// TIA Portal V20 export
// export: Created 2026-04-11T06:02:30.0272566Z, ExportSetting WithDefaults, DisplayName Totally Integrated Automation Portal, DisplayVersion V20, DisplayName TIA Portal Openness, DisplayVersion V20, DisplayName TIA Portal Version Control Interface, DisplayVersion V20, DisplayName STEP 7 Professional, DisplayVersion V20, DisplayName STEP 7 Safety, DisplayVersion V20, DisplayName WinCC Basic/Comfort/Advanced, DisplayVersion V20, DisplayName WinCC Unified, DisplayVersion V20
TYPE "udtError_MicroMotion"
// stored: IsFailsafeCompliant false
   STRUCT
      ResetFailed { ExternalWritable := 'False'} : Bool;   // Can't reset MicroMotion
      FlowWithoutRequest { ExternalWritable := 'False'} : Bool;   // Flow detected, but no request
   END_STRUCT;
END_TYPE
